TYPE STU_Part :
STRUCT
	user1	: BOOL;
	user2	: BOOL;
	user3	: INT;
	user4	: INT;	
END_STRUCT
END_TYPE

(* stored: Version 1.1.0.1
   DUT STU_Part: Id {a3e0cd40-cdf8-483c-8df6-59575a72bd5f} *)
